// TwinCAT 3 PLC project Untitled1
// ProgramVersion: 3.1.4023.0
// libraries:
//   Tc2_SerialCom, * (Beckhoff Automation GmbH)
//   Tc2_Standard, * (Beckhoff Automation GmbH)
//   Tc2_System, * (Beckhoff Automation GmbH)
//   Tc3_Module, * (Beckhoff Automation GmbH)
// project tree:
//   GVLs/ GVL.TcGVL
//   POUs/ BackgroundEL.TcPOU, MAIN.TcPOU
//   / Task_COM.TcTTO

CONFIGURATION Untitled1
    RESOURCE PLC ON TwinCAT3
        TASK Task_COM(INTERVAL := T#125us, PRIORITY := 61);
        PROGRAM BackgroundEL WITH Task_COM : BackgroundEL;
    END_RESOURCE
END_CONFIGURATION

// ---- GVLs/GVL.TcGVL
VAR_GLOBAL
	RxBufferEL			: ComBuffer;	(* Receive data buffer; used with all receive function blocks *)
	TxBufferEL			: ComBuffer;	(* Transmit data buffer; used with all receive function blocks *)

END_VAR

// ---- POUs/BackgroundEL.TcPOU
PROGRAM BackgroundEL
VAR
	(* background communication with the EL6001 terminal *)
	fbEL6022Ctrl		: SerialLineControl;
	bEL6022CtrlError	: BOOL;
	eEL6022CtrlErrorID	: ComError_t;
	(* 	I/O variables for a EL6001 terminal*)
	stIn_EL6022 AT %I*	: EL6inData22B;	(* linked to the EL6001 in the TwinCAT System Manager *)
	stOut_EL6022 AT %Q*	: EL6outData22B;(* linked to the EL6001 in the TwinCAT System Manager *)
END_VAR

(*
The SerialLineControl function block is supposed to be called in every PLC cycle.
It communicates with the serial line hardware device and transmits or receives data.
The SerialLineControl can be called in the standard task (e.g.for PcCOM port usage) 
or in a separate fast task (e.g.for terminal usage) as well.
A fast separate task will be necessary at high baud rates or with KL6001 terminals 
which have a small process image (3 or 5 data bytes only)
*)

(* background communication with the EL6001 terminal *)
fbEL6022Ctrl(
	Mode:= SERIALLINEMODE_EL6_22B, 
	pComIn:= ADR(stIn_EL6022), 
	pComOut:= ADR(stOut_EL6022), 
	SizeComIn:= SIZEOF(stIn_EL6022), 
	Error=> , 
	ErrorID=> , 
	TxBuffer:= TxBufferEL, 
	RxBuffer:= RxBufferEL );
IF fbEL6022Ctrl.Error THEN
	bEL6022CtrlError := TRUE;
	eEL6022CtrlErrorID := fbEL6022Ctrl.ErrorID;
END_IF

END_PROGRAM

// ---- POUs/MAIN.TcPOU
PROGRAM MAIN

VAR
	case_var : INT := 0;
	Timer		: TON := (PT:=T#1MS);

	fbReceive		: ReceiveString;
	sReceivedString	: STRING;
	sLastReceivedString: STRING;
	sCleanedLastReceivedString: STRING;
	bStringReceived	: BOOL;
	bReceiveBusy	: BOOL;
	bReceiveError	: BOOL;
	eReceiveErrorID	: ComError_t;
	bReceiveTimeout	: BOOL;
	nReceiveCounter	: UDINT;
	cleanedLastReceivedString: STRING;
END_VAR

VAR_OUTPUT
	fWeightInKG AT %Q* : REAL;
END_VAR

CASE case_var OF

0:
	Timer(IN:=TRUE);
	IF Timer.Q THEN
		Timer(IN:=FALSE); (* reset timer *)
		case_var := 1;
	END_IF

1:
fbReceive(
	Prefix:= '',
	Suffix:= '$0D$0A',
	ReceivedString:= sReceivedString,
	RXbuffer:= RxBufferEL,
	StringReceived=> bStringReceived,
	Busy=> bReceiveBusy,
	Error=> ,
	RxTimeout=> bReceiveTimeout );
IF fbReceive.Error <> COMERROR_NOERROR THEN
	eReceiveErrorID := fbReceive.Error;
END_IF
IF bStringReceived THEN
	case_var := 0;
	nReceiveCounter := nReceiveCounter + 1;
	sLastReceivedString := sReceivedString;
	sCleanedLastReceivedString := DELETE(sLastReceivedString, 2, 7);
	fWeightInKG := STRING_TO_REAL(sCleanedLastReceivedString) / 1000;
END_IF
END_CASE

END_PROGRAM
